{attribute 'qualified_only'}
VAR_GLOBAL
	startButton	:	NormallyOpenPushButton;
	stopButton	:	NormallyClosedPushButton;
	emergencyStopButton	:	NormallyClosedPushButton;
	productDetectedSensor	:	NormallyClosedSensor;
	conveyorFullSensor	:	NormallyClosedSensor;
	backupConveyorFullSensor	:	NormallyClosedSensor;
	conveyorMotor	:	DirectOnlineStarterMotor;
	
	sortingConveyor	:	SortingConveyor(ProductDetected := productDetectedSensor,
		                                ConveyorFull := conveyorFullSensor,
										ConveyorMotor := conveyorMotor);
	
	myConveyorSortingMachine	:	MyConveyorSortingMachine( StartButton := startButton,
                                                              StopButton := stopButton,
															  EmergencyStopButton := emergencyStopButton,
															  ConveyorModule := sortingConveyor);
END_VAR

(* stored: Version 1.1.0.1, ProductVersion 3.1.4024.11
   GVL GVL: Id {788d73b2-c2a2-47f5-ab0a-e80d75f6a820} *)
